FUNCTION_BLOCK App2_StripperTempandStripperLevelandProdRate (* Composite Function Block Type *)
  (* Standard: 61499-2 *)
  (* Version 0.0, 2018-11-06, 4DIAC-IDE, 4DIAC-Consortium *)
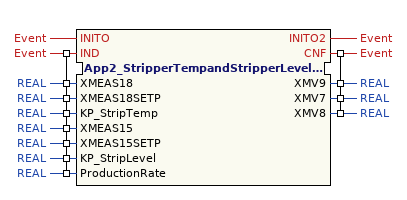
  EVENT_INPUT
    INITO; (* Initialization Request *)
    IND WITH XMEAS18, XMEAS18SETP, XMEAS15, XMEAS15SETP, KP_StripTemp, KP_StripLevel, ProductionRate; (* Normal Execution Request *)
  END_EVENT
  EVENT_OUTPUT
    INITO2; (* Initialization Confirm *)
    CNF WITH XMV9, XMV7, XMV8; (* Execution Confirmation *)
  END_EVENT
  VAR_INPUT
    XMEAS18 : REAL;
    XMEAS18SETP : REAL;
    KP_StripTemp : REAL;
    XMEAS15 : REAL;
    XMEAS15SETP : REAL;
    KP_StripLevel : REAL;
    ProductionRate : REAL;
  END_VAR
  VAR_OUTPUT
    XMV9 : REAL;
    XMV7 : REAL;
    XMV8 : REAL;
  END_VAR
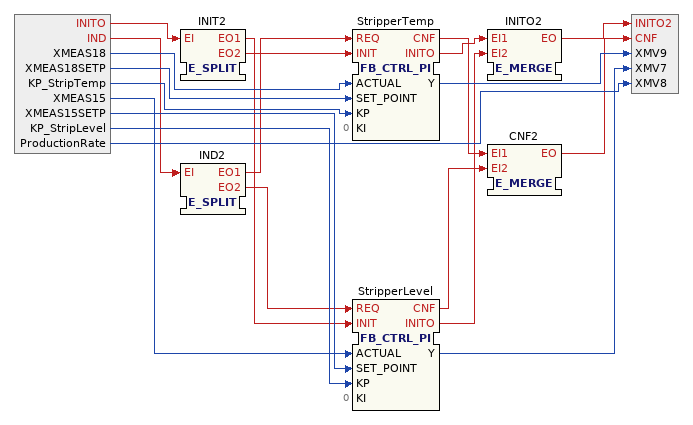
  FBS
    IND2 : E_SPLIT;
    StripperTemp : FB_CTRL_PI(KI := 0);
    StripperLevel : FB_CTRL_PI(KI := 0);
    CNF2 : E_MERGE;
    INIT2 : E_SPLIT;
    INITO2 : E_MERGE;
  END_FBS
  EVENT_CONNECTIONS
    IND2.EO1 TO StripperTemp.REQ;
    IND2.EO2 TO StripperLevel.REQ;
    StripperTemp.CNF TO CNF2.EI1;
    StripperLevel.CNF TO CNF2.EI2;
    CNF2.EO TO CNF;
    IND TO IND2.EI;
    INITO TO INIT2.EI;
    INIT2.EO1 TO StripperTemp.INIT;
    INIT2.EO2 TO StripperLevel.INIT;
    StripperTemp.INITO TO INITO2.EI1;
    StripperLevel.INITO TO INITO2.EI2;
    INITO2.EO TO INITO2;
  END_CONNECTIONS
  DATA_CONNECTIONS
    StripperTemp.Y TO XMV9;
    StripperLevel.Y TO XMV7;
    XMEAS18 TO StripperTemp.ACTUAL;
    XMEAS18SETP TO StripperTemp.SET_POINT;
    XMEAS15 TO StripperLevel.ACTUAL;
    XMEAS15SETP TO StripperLevel.SET_POINT;
    KP_StripTemp TO StripperTemp.KP;
    KP_StripLevel TO StripperLevel.KP;
    ProductionRate TO XMV8;
  END_CONNECTIONS
END_FUNCTION_BLOCK
